// TIA Portal V19 export
TYPE "LEXCHANGETRAY_typeConstraintRollerEm_interface"
// stored: Access Published
   STRUCT
      deliver : "LEXCHANGETRAY_typeConstraintRollerEm_deliver_interface";
      recieve : "LEXCHANGETRAY_typeConstraintRollerEm_recieve_interface";
   END_STRUCT;
END_TYPE
